// TIA Portal V19 export
FUNCTION_BLOCK "LAF_ManageAlarms"   // FB82, LAD
TITLE = LAF_ManageAlarms
AUTHOR : Siemens Digital Industries
FAMILY : LAF
VERSION : 1.2
// Mapping the ProDiag categories to the commands of the ModeStateManager.
// stored: Access Published, IsIECCheckEnabled true, MemoryReserve 100, SetENOAutomatically true
   VAR_INPUT
      proDiagState : SV_FB_State_V2;   // ProDiag DB
   END_VAR
   VAR_OUTPUT
      parentAlarmDB { ExternalWritable := 'False'} : "LAF_typeAlarms";
      alarmDB { ExternalWritable := 'False'} : "LAF_typeAlarms";
      hmiInterfaceDB { ExternalWritable := 'False'} : "LAF_typeAlarms";
   END_VAR
   VAR_IN_OUT
      commands : "LUC_typeStateCommands";
   END_VAR
BEGIN

REGION Network 1: BLOCK INFO HEADER
   // SIEMENS AG / (c)Copyright 2024
   // ------------------------------------------------------------------------------
   // Title:            LAF_ManageAlarms
   // Comment/Function: Mapping the ProDiag categories to the commands of the ModeStateManager.
   // Library/Family:   Library of Automation Framework
   // Author:                Siemens Digital Industry
   // Tested with:       S7-PLCSIM Advanced 6.0
   // Engineering:      TIA Portal V19
   // Restrictions:       ---
   // Requirements:   ---
   // ------------------------------------------------------------------------------
   // Change log table:
   // Version  | Date       | Expert in charge       | Changes applied
   // ---------|------------|------------------------|------------------------------
   // 01.01.00 | 21.06.2024 | SIMATIC Systems Support
   //                         First released version
   // 01.02.00 | 30.09.2024 | SIMATIC Systems Support
   //                         Block information properties updated
END_REGION

REGION Network 2: Stop command
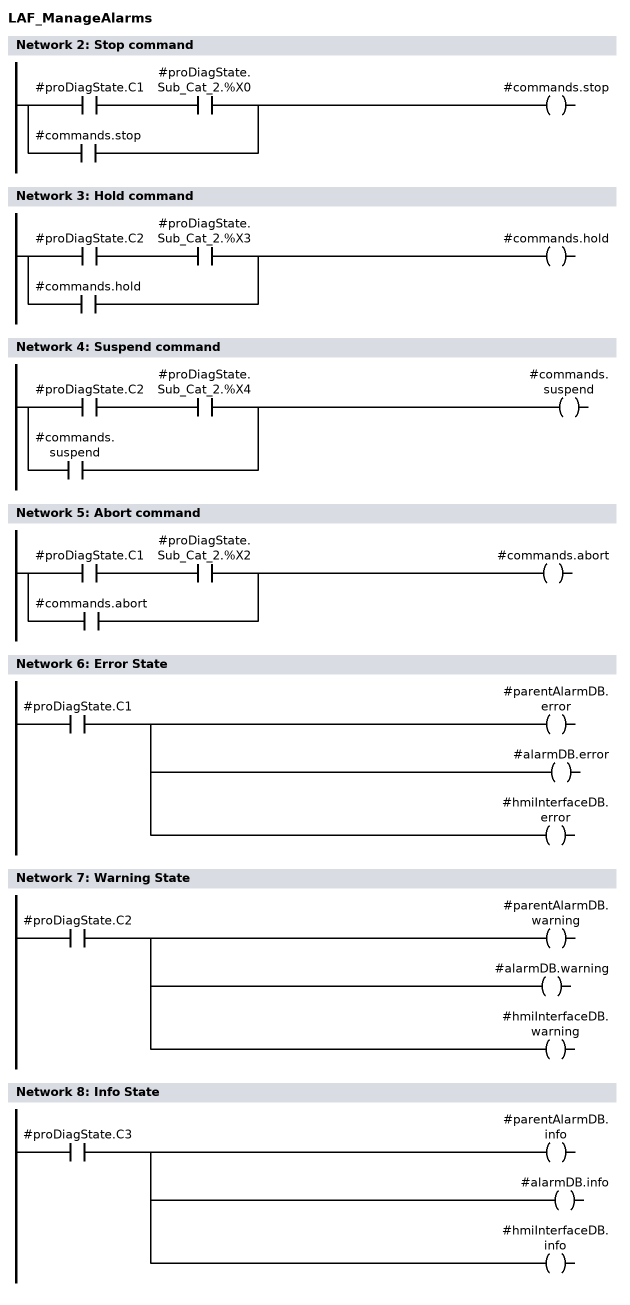
   RUNG wire#powerrail
      Contact( #proDiagState.C1 )
      Contact( #proDiagState.Sub_Cat_2.%X0 )
      wire#w1
      Coil( #commands.stop )
   END_RUNG
   RUNG wire#powerrail
      Contact( #commands.stop )
   END_RUNG wire#w1
   // the same network as SCL:
   #commands.stop := (#proDiagState.C1 AND #proDiagState.Sub_Cat_2.%X0) OR #commands.stop;
END_REGION

REGION Network 3: Hold command
   RUNG wire#powerrail
      Contact( #proDiagState.C2 )
      Contact( #proDiagState.Sub_Cat_2.%X3 )
      wire#w1
      Coil( #commands.hold )
   END_RUNG
   RUNG wire#powerrail
      Contact( #commands.hold )
   END_RUNG wire#w1
   // the same network as SCL:
   #commands.hold := (#proDiagState.C2 AND #proDiagState.Sub_Cat_2.%X3) OR #commands.hold;
END_REGION

REGION Network 4: Suspend command
   RUNG wire#powerrail
      Contact( #proDiagState.C2 )
      Contact( #proDiagState.Sub_Cat_2.%X4 )
      wire#w1
      Coil( #commands.suspend )
   END_RUNG
   RUNG wire#powerrail
      Contact( #commands.suspend )
   END_RUNG wire#w1
   // the same network as SCL:
   #commands.suspend := (#proDiagState.C2 AND #proDiagState.Sub_Cat_2.%X4) OR #commands.suspend;
END_REGION

REGION Network 5: Abort command
   RUNG wire#powerrail
      Contact( #proDiagState.C1 )
      Contact( #proDiagState.Sub_Cat_2.%X2 )
      wire#w1
      Coil( #commands.abort )
   END_RUNG
   RUNG wire#powerrail
      Contact( #commands.abort )
   END_RUNG wire#w1
   // the same network as SCL:
   #commands.abort := (#proDiagState.C1 AND #proDiagState.Sub_Cat_2.%X2) OR #commands.abort;
END_REGION

REGION Network 6: Error State
   RUNG wire#powerrail
      Contact( #proDiagState.C1 )
      wire#w1
      Coil( #parentAlarmDB.error )
   END_RUNG
   RUNG wire#w1
      Coil( #alarmDB.error )
   END_RUNG
   RUNG wire#w1
      Coil( #hmiInterfaceDB.error )
   END_RUNG
   // the same network as SCL:
   #parentAlarmDB.error := #proDiagState.C1;
   #alarmDB.error := #proDiagState.C1;
   #hmiInterfaceDB.error := #proDiagState.C1;
END_REGION

REGION Network 7: Warning State
   RUNG wire#powerrail
      Contact( #proDiagState.C2 )
      wire#w1
      Coil( #parentAlarmDB.warning )
   END_RUNG
   RUNG wire#w1
      Coil( #alarmDB.warning )
   END_RUNG
   RUNG wire#w1
      Coil( #hmiInterfaceDB.warning )
   END_RUNG
   // the same network as SCL:
   #parentAlarmDB.warning := #proDiagState.C2;
   #alarmDB.warning := #proDiagState.C2;
   #hmiInterfaceDB.warning := #proDiagState.C2;
END_REGION

REGION Network 8: Info State
   RUNG wire#powerrail
      Contact( #proDiagState.C3 )
      wire#w1
      Coil( #parentAlarmDB.info )
   END_RUNG
   RUNG wire#w1
      Coil( #alarmDB.info )
   END_RUNG
   RUNG wire#w1
      Coil( #hmiInterfaceDB.info )
   END_RUNG
   // the same network as SCL:
   #parentAlarmDB.info := #proDiagState.C3;
   #alarmDB.info := #proDiagState.C3;
   #hmiInterfaceDB.info := #proDiagState.C3;
END_REGION
END_FUNCTION_BLOCK
